// TIA Portal V19 export
DATA_BLOCK "MixingIngredientsBread"   // DB206
// stored: MemoryReserve 100
   VAR
      mixingBread { S7_SetPoint := 'True'} : "typeMixinIngredientsBread";
   END_VAR
BEGIN
END_DATA_BLOCK
